FUNCTION_BLOCK PI_REAL
  (* Standard: 61499-2 *)
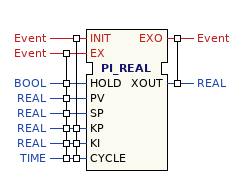
  EVENT_INPUT
    INIT WITH KP, KI, CYCLE;
    EX WITH HOLD, PV, SP, KP, KI, CYCLE;
  END_EVENT
  EVENT_OUTPUT
    EXO WITH XOUT;
  END_EVENT
  VAR_INPUT
    HOLD : BOOL;
    PV : REAL;
    SP : REAL;
    KP : REAL;
    KI : REAL;
    CYCLE : TIME;
  END_VAR
  VAR_OUTPUT
    XOUT : REAL;
  END_VAR
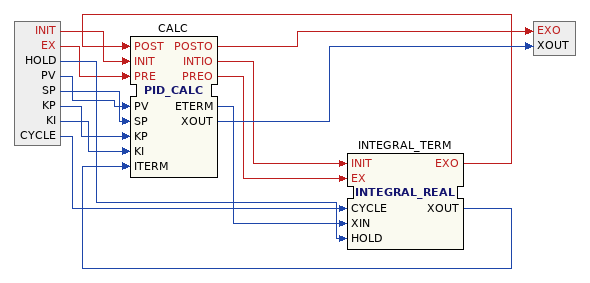
  FBS
    CALC : PID_CALC;
    INTEGRAL_TERM : INTEGRAL_REAL;
  END_FBS
  EVENT_CONNECTIONS
    CALC.POSTO TO EXO;
    CALC.INTIO TO INTEGRAL_TERM.INIT;
    CALC.PREO TO INTEGRAL_TERM.EX;
    INTEGRAL_TERM.EXO TO CALC.POST;
    INIT TO CALC.INIT;
    EX TO CALC.PRE;
  END_CONNECTIONS
  DATA_CONNECTIONS
    PV TO CALC.PV;
    SP TO CALC.SP;
    KP TO CALC.KP;
    KI TO CALC.KI;
    CYCLE TO INTEGRAL_TERM.CYCLE;
    CALC.ETERM TO INTEGRAL_TERM.XIN;
    CALC.XOUT TO XOUT;
    INTEGRAL_TERM.XOUT TO CALC.ITERM;
    HOLD TO INTEGRAL_TERM.HOLD;
  END_CONNECTIONS
END_FUNCTION_BLOCK
